TYPE teCTCEvent :
(
	CTC_NO_EVENT 					:= 0,
	CTC_EVENT_UNDERTEMP_MC 			:= 6210,
	CTC_EVENT_OVERTEMP_MC 			:= 6211,
	CTC_EVENT_UNDERTEMP_CB 			:= 6212,
	CTC_EVENT_OVERTEMP_CB 			:= 6213,
	CTC_EVENT_UNDERTEMP_EB 			:= 6214,
	CTC_EVENT_OVERTEMP_EB 			:= 6215,
	CTC_EVENT_OVERTEMP_PS_PHASE_U 	:= 6216,
	CTC_EVENT_OVERTEMP_PS_PHASE_V 	:= 6217,
	CTC_EVENT_OVERTEMP_PS_PHASE_W 	:= 6218,
	CTC_EVENT_OVERTEMP_MOT_PHASE_U 	:= 6219,
	CTC_EVENT_OVERTEMP_MOT_PHASE_V 	:= 6220,
	CTC_EVENT_OVERTEMP_MOT_PHASE_W 	:= 6221,
	CTC_EVENT_CONTROLLER_ERROR 		:= 6222,
	CTC_EVENT_INTERNAL_ERROR 		:= 6223,
	CTC_EVENT_TRACKING_ERROR 		:= 6224,
	CTC_EVENT_INVALID_SETPOINTS 	:= 6225,
	CTC_EVENT_OVERVOLTAGE_LOGIC 	:= 20752,
	CTC_EVENT_UNDERVOLTAGE_LOGIC 	:= 20753,
	CTC_EVENT_OVERVOLTAGE_POWER 	:= 20754,
	CTC_EVENT_HOMING_FAILED 		:= 6226
);
END_TYPE

(* stored: Version 1.1.0.1, ProductVersion 3.1.4026.17
   EnumerationTextList teCTCEvent: Id {09772d6b-33b3-4495-b7cf-3fb878e5632f} *)
